DATA_BLOCK "Positionen"
TITLE = Positionswerte
VERSION : 0.1


  STRUCT
   Pos1 : INT  := 78;	//Ablagepostion Kunststoffteile und  Metallteile ohne Bohrung
   Pos2 : INT  := 53;	//Ablageposition Metallteile mit Bohrung
   Pos3 : INT  := 31;	//Reserve Position
   Pos4 : INT  := 6;	//Reserve Position
  END_STRUCT ;
BEGIN

END_DATA_BLOCK

